// Mitsubishi GX Works2 project: factory   PLC: Q02/Q02H

PROGRAM MAIN
VAR
  cy_1 : cy;
  cy_2 : cy;
  cy_3 : cy;
END_VAR
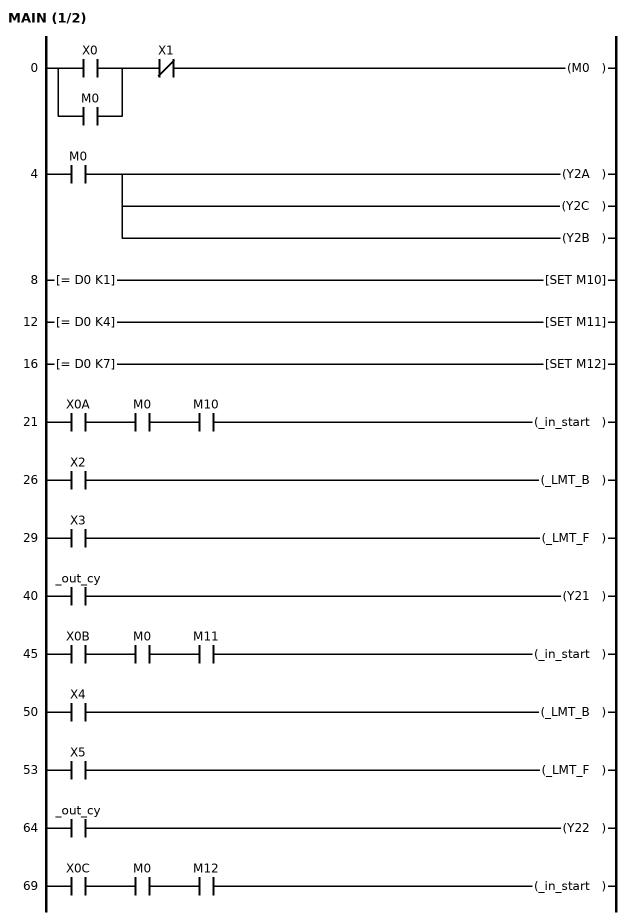
0     LD      X0
      OR      M0
      ANI     X1
      OUT     M0
4     LD      M0
      OUT     Y2A
      OUT     Y2C
      OUT     Y2B
8     LD=     D0 K1
      SET     M10
12    LD=     D0 K4
      SET     M11
16    LD=     D0 K7
      SET     M12
; FB BLK START cy(cy_1)
21    LD      X0A
      AND     M0
      AND     M10
      OUT     _in_start
26    LD      X2
      OUT     _LMT_B
29    LD      X3
      OUT     _LMT_F
; FB START
; FB_NAME cy
; INSTANCE_NAME cy_1
; FB IN_B:in_start
; FB OUT_out_cy:B
; FB IN_B:LMT_B
; FB IN_B:LMT_F
; FB END
40    LD      _out_cy
      OUT     Y21
; FB BLK END
; FB BLK START cy(cy_2)
45    LD      X0B
      AND     M0
      AND     M11
      OUT     _in_start
50    LD      X4
      OUT     _LMT_B
53    LD      X5
      OUT     _LMT_F
; FB START
; FB_NAME cy
; INSTANCE_NAME cy_2
; FB IN_B:in_start
; FB OUT_out_cy:B
; FB IN_B:LMT_B
; FB IN_B:LMT_F
; FB END
64    LD      _out_cy
      OUT     Y22
; FB BLK END
; FB BLK START cy(cy_3)
69    LD      X0C
      AND     M0
      AND     M12
      OUT     _in_start
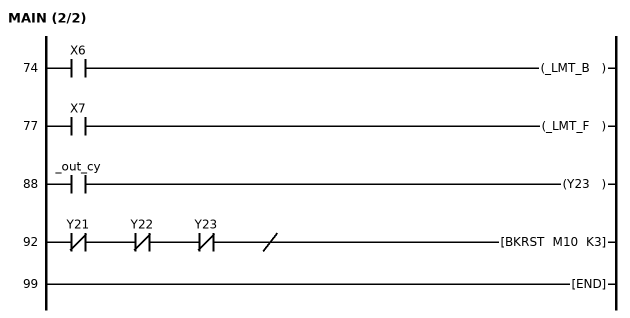
74    LD      X6
      OUT     _LMT_B
77    LD      X7
      OUT     _LMT_F
; FB START
; FB_NAME cy
; INSTANCE_NAME cy_3
; FB IN_B:in_start
; FB OUT_out_cy:B
; FB IN_B:LMT_B
; FB IN_B:LMT_F
; FB END
88    LD      _out_cy
      OUT     Y23
; FB BLK END
92    LDI     Y21
      ANI     Y22
      ANI     Y23
      INV
      BKRST   M10 K3
99    END
END_PROGRAM

FUNCTION_BLOCK cy
VAR_INPUT
  in_start : BOOL;
END_VAR
VAR
  mem0 : BOOL;
  FT0 : TIMER;
END_VAR
VAR_INPUT
  LMT_B : BOOL;
END_VAR
VAR_OUTPUT
  out_cy : BOOL;
END_VAR
VAR_INPUT
  LMT_F : BOOL;
END_VAR
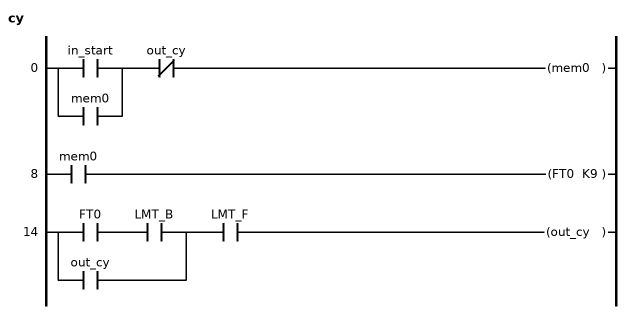
0     LD      in_start
      OR      mem0
      ANI     out_cy
      OUT     mem0
8     LD      mem0
      OUT     FT0 K9
14    LD      FT0
      AND     LMT_B
      OR      out_cy
      AND     LMT_F
      OUT     out_cy
END_FUNCTION_BLOCK
